PROGRAM STATION1
VAR

	tDelay: TON;
	bDELAY: BOOL:=FALSE;
END_VAR

tDelay(IN:=bDELAY);
CASE eSTATION1_STATE OF
	E_STATION_STATE.uninit:
		eSTATION1_STATE:= E_STATION_STATE.idle;

	E_STATION_STATE.idle:
		bS1_RUNNING:=FALSE;
			

	E_STATION_STATE.do_action1://delay and open piston1,2
		tDELAY.PT:=T#1S;
		bDELAY:=TRUE;
		IF tDELAY.Q THEN
			bDELAY:=FALSE;
			fbPISTON[1].A_OPEN();
			fbPISTON[2].A_OPEN();
		END_IF
		
		IF fbPISTON[1].PistonStatus= ePistonStatus.OPENED  AND fbPISTON[2].PistonStatus= ePistonStatus.OPENED THEN
			eSTATION1_STATE:=E_STATION_STATE.do_action2;
		END_IF
		
	E_STATION_STATE.do_action2://delay and close pistons 1,2
		tDELAY.PT:=T#2S;		
		bDELAY:=TRUE;
		IF tDELAY.Q THEN
			bDELAY:=FALSE;
			fbPISTON[1].A_CLOSE();
			fbPISTON[2].A_CLOSE();
		END_IF
		IF fbPISTON[1].PistonStatus= ePistonStatus.CLOSED  AND fbPISTON[2].PistonStatus= ePistonStatus.CLOSED THEN
			eSTATION1_STATE:=E_STATION_STATE.do_action3;
		END_IF
	
	E_STATION_STATE.do_action3://delay and open piston 3
		tDELAY.PT:=T#2S;
		bDELAY:=TRUE;
		IF tDELAY.Q THEN
			bDELAY:=FALSE;
			fbPISTON[3].A_OPEN();
		END_IF
		
		IF fbPISTON[3].PistonStatus= ePistonStatus.OPENED THEN
			eSTATION1_STATE:=E_STATION_STATE.do_action4;
		END_IF
	
	E_STATION_STATE.do_action4://delay and close pistons 1,2
		tDELAY.PT:=T#2S;		
		bDELAY:=TRUE;
		IF tDELAY.Q THEN
			bDELAY:=FALSE;
			fbPISTON[3].A_CLOSE();
		END_IF
		IF fbPISTON[3].PistonStatus= ePistonStatus.CLOSED  THEN
			eSTATION1_STATE:=E_STATION_STATE.do_action5;
		END_IF
		
	E_STATION_STATE.do_action5://delay 
		tDELAY.PT:=T#2S;
		bDELAY:=TRUE;
		IF tDELAY.Q THEN
			bDELAY:=FALSE;
			eSTATION1_STATE:=E_STATION_STATE.done;
		END_IF
	
	E_STATION_STATE.done:
		bS1_RUNNING:=FALSE;

END_CASE

END_PROGRAM

(* stored: Version 1.1.0.1, ProductVersion 3.1.4024.12
   POU STATION1: Id {118c21d3-d07f-48b2-af87-ee9537ae1c73}, SpecialFunc None *)
